// TIA Portal V19 export
TYPE "LAF_typeConstraintWorkstationEm3ParametersInterfaceHmi"
// stored: Access Published
   STRUCT
      configuration : "LAF_typeConstraintWorkstationEm3ParametersHmi";
      commands : "LBC_typeInterfaceCommands";
      monitoring { S7_SetPoint := 'True'} : "LAF_typeConstraintWorkstationEm3ProcessValuesHmi";
   END_STRUCT;
END_TYPE
